// TwinCAT 3 PLC project PLC_Project
// ProgramVersion: 3.1.4023.0
// libraries:
//   Tc2_EtherCAT, * (Beckhoff Automation GmbH)
//   Tc2_Standard, * (Beckhoff Automation GmbH)
//   Tc2_System, * (Beckhoff Automation GmbH)
//   Tc3_Module, * (Beckhoff Automation GmbH)
// project tree:
//   DUTs/EA_Device_IO/Helpers/ ST_AdsAddr.TcDUT, ST_EA_InfoData.TcDUT, ST_EA_RxPDO.TcDUT, ST_EA_TxPDO.TcDUT
//   DUTs/EA_Device_IO/ ST_EA_IO.TcDUT
//   / PlcTask.TcTTO
//   POUs/Function Blocks/ FB_EA_Interface.TcPOU
//   POUs/ MAIN.TcPOU
// real-time tasks:
//   TASK PlcTask: cycle T#10ms, priority 20, ADS port 350
// I/O:
//   DEVICE Device 1 (EtherCAT), AmsNetId 192.168.42.20.2.1
//     Box 1 (IF-AB-ECT for standard) [IF-AB-ECT for standard]
// variable links:
//   PLC_Project/PLC_Project Instance <-> Device 1 (EtherCAT)/Box 1 (IF-AB-ECT for standard)
//     PlcTask Inputs/MAIN.fbEAInterface[1].stHWVar.stInfoData @bit 16 <-> InfoData/AdsAddr
//     PlcTask Inputs/MAIN.fbEAInterface[1].stHWVar.stInfoData <-> InfoData/State
//     PlcTask Inputs/MAIN.fbEAInterface[1].stHWVar.stRxPDO @bit 64 <-> DO RxPDO-Map/Control
//     PlcTask Inputs/MAIN.fbEAInterface[1].stHWVar.stRxPDO @bit 48 <-> DO RxPDO-Map/Current monitor
//     PlcTask Inputs/MAIN.fbEAInterface[1].stHWVar.stRxPDO @bit 112 <-> DO RxPDO-Map/Current select
//     PlcTask Inputs/MAIN.fbEAInterface[1].stHWVar.stRxPDO @bit 128 <-> DO RxPDO-Map/Power select
//     PlcTask Inputs/MAIN.fbEAInterface[1].stHWVar.stRxPDO @bit 144 <-> DO RxPDO-Map/Resistance select
//     PlcTask Inputs/MAIN.fbEAInterface[1].stHWVar.stRxPDO <-> DO RxPDO-Map/Status
//     PlcTask Inputs/MAIN.fbEAInterface[1].stHWVar.stRxPDO @bit 32 <-> DO RxPDO-Map/Voltage monitor
//     PlcTask Inputs/MAIN.fbEAInterface[1].stHWVar.stRxPDO @bit 96 <-> DO RxPDO-Map/Voltage select
//     PlcTask Outputs/MAIN.fbEAInterface[1].stHWVar.stTxPDO @bit 16 <-> DI TxPDO-Map/Current select
//     PlcTask Outputs/MAIN.fbEAInterface[1].stHWVar.stTxPDO @bit 32 <-> DI TxPDO-Map/Power select
//     PlcTask Outputs/MAIN.fbEAInterface[1].stHWVar.stTxPDO @bit 48 <-> DI TxPDO-Map/Resistance select
//     PlcTask Outputs/MAIN.fbEAInterface[1].stHWVar.stTxPDO <-> DI TxPDO-Map/Voltage select

CONFIGURATION PLC_Project
    RESOURCE PLC ON TwinCAT3
        TASK PlcTask(INTERVAL := T#10ms, PRIORITY := 20);
        PROGRAM MAIN WITH PlcTask : MAIN;
    END_RESOURCE
END_CONFIGURATION

// ---- DUTs/EA_Device_IO/Helpers/ST_AdsAddr.TcDUT
TYPE ST_AdsAddr :
STRUCT
	netID		: AMSNETID;
	port		: WORD;
END_STRUCT
END_TYPE

// ---- DUTs/EA_Device_IO/Helpers/ST_EA_InfoData.TcDUT
TYPE ST_EA_InfoData :
STRUCT
	nState				: UINT;
	stAdsAddr			: ST_AdsAddr;
END_STRUCT
END_TYPE

// ---- DUTs/EA_Device_IO/Helpers/ST_EA_RxPDO.TcDUT
TYPE ST_EA_RxPDO :
STRUCT
	nStatus			 : UDINT;
	nVoltageMon		 : UINT;
	nCurrentMon		 : UINT;
	nControl		 : UDINT;
	nVoltageSel		 : UINT;
	nCurrentSel		 : UINT;
	nPowerSel		 : UINT;
	nResistanceSel	 : UINT;
END_STRUCT
END_TYPE

// ---- DUTs/EA_Device_IO/Helpers/ST_EA_TxPDO.TcDUT
TYPE ST_EA_TxPDO :
STRUCT
	nVoltageSel 		:	UINT;
	nCurrentSel			: 	UINT;
	nPowerSel			: 	UINT;
	nResistanceSel		: 	UINT;
END_STRUCT
END_TYPE

// ---- DUTs/EA_Device_IO/ST_EA_IO.TcDUT
TYPE ST_EA_IO :
STRUCT
	stRxPDO			AT%I* 	: ST_EA_RxPDO;
	stTxPDO			AT%Q* 	: ST_EA_TxPDO;
	stInfoData		AT%I* 	: ST_EA_InfoData;
END_STRUCT
END_TYPE

// ---- POUs/MAIN.TcPOU
PROGRAM MAIN
VAR CONSTANT
	CONST_MAX_NUMBER_OF_EA_DEVICES	: INT:= 1;
END_VAR

VAR
	fbEAInterface					: ARRAY [1..CONST_MAX_NUMBER_OF_EA_DEVICES] OF FB_EA_Interface;
	nDeviceIdx						: INT	:= 1;
END_VAR


FOR nDeviceIdx := 1 TO CONST_MAX_NUMBER_OF_EA_DEVICES DO
	
	fbEAInterface[nDeviceIdx]();


END_FOR

END_PROGRAM

// ---- POUs/Function Blocks/FB_EA_Interface.TcPOU
FUNCTION_BLOCK FB_EA_Interface
VAR_INPUT
	//Device Specifications - From Datasheet of the PSU/Load
	rMax_Current					: REAL;							
	rMax_Voltage					: REAL;
	rMax_Power						: REAL;
	rMax_Resistance					: REAL;
	
	//Setpoint
	rCurrent_Setpoint				: REAL;
	rVoltage_Setpoint				: REAL;
	rPower_Setpoint					: REAL;
	rResistance_Setpoint			: REAL;
	
	bRemote							: BOOL 		:= TRUE;
	bPowerStage						: BOOL;
END_VAR
VAR_OUTPUT
	bRemoteStatus					: BOOL;
	bPowerStageStatus				: BOOL;
	
	rCurrent_Actual					: REAL;
	rVoltage_Actual					: REAL;	
END_VAR
VAR
	stHWVar							: ST_EA_IO;
	                				
	eState							: (INIT, AUTO_ON, REMOTE, IDLE, POWER_STAGE_ON, POWER_STAGE_OFF, DONE, ERROR);  
	eParam							: (AUTO_ON,POWER_ON,REMOTE,POWER_STAGE);
	
	fbWriteCoe						: FB_ECCoeSdoWriteEx;
	
	nCoEVal							: ARRAY [1..4] OF UINT;
	bAutoOn							: BOOL;
	
END_VAR

VAR CONSTANT
	//CoE Index
	
	nCoeIdx_Remote					: WORD		:= 16#2193;
	nCoeIdx_AutoOn					: WORD		:= 16#2198;
	nCoeIdx_PowerOn					: WORD		:= 16#2199;
	nCoeIdx_PowerStage				: WORD		:= 16#2196;
		
END_VAR


ACT_Scaling();

CASE eState OF
	
	INIT: 
	
		fbWriteCoe(
			bExecute				:= FALSE);
			
				
		nCoEVal[AUTO_ON]			:= 65280;
		nCoEVal[POWER_ON]			:= 65535;
		nCoEVal[REMOTE]				:= 65280;
		nCoEVal[POWER_STAGE]		:= 0;
		
		IF NOT fbWriteCoe.bBusy
		AND stHWVar.stInfoData.nState=8						//Device in OP
		THEN
		
			eState					:= AUTO_ON;
			
		END_IF
					
			
	AUTO_ON:
	
		IF NOT fbWriteCoe.bBusy
		THEN
			ACT_AutoOn();
		ELSE
			eState					:= POWER_ON;
		END_IF
	
		
	
		
END_CASE

ACTION ACT_Auto_On:

END_ACTION

ACTION ACT_AutoOn:


fbWriteCoe(
	sNetID			:= stHWVar.stInfoData.stAdsAddr.netID,
	nSlaveAddr		:= stHWVar.stInfoData.stAdsAddr.port,
	nIndex			:= nCoeIdx_AutoOn,
	pSrcBuf			:= ADR(nCoEVal[AUTO_ON]),
	cbBufLen		:= SIZEOF(nCoeVal[AUTO_ON]),
	bExecute		:= TRUE);
END_ACTION

ACTION ACT_Scaling:


//Setpoint Scaling

stHWVar.stTxPDO.nCurrentSel			:= REAL_TO_UINT(rCurrent_Setpoint 	* (rMax_Current/65535));
stHWVar.stTxPDO.nPowerSel			:= REAL_TO_UINT(rPower_Setpoint 	* (rMax_Power/65535));
stHWVar.stTxPDO.nVoltageSel			:= REAL_TO_UINT(rVoltage_Setpoint 	* (rMax_Voltage/65535));
stHWVar.stTxPDO.nResistanceSel		:= REAL_TO_UINT(rResistance_Setpoint* (rMax_Resistance/65535));

//Actual Value Scaling


rCurrent_Actual						:= stHWVar.stRxPDO.nCurrentMon	/ rMax_Current;
rVoltage_Actual						:= stHWVar.stRxPDO.nVoltageMon	/ rMax_Voltage;
END_ACTION

END_FUNCTION_BLOCK
